{attribute 'qualified_only'}
{attribute 'strict'}
TYPE E_InputTransportTube :
(
	BI1 := 0
) UINT;
END_TYPE

(* stored: Version 1.1.0.1, ProductVersion 3.1.4022.17
   DUT E_InputTransportTube: Id {26e13819-1baa-4350-8f0d-08839603bdb0} *)
